# EPICS autosave request: iocBoot/iocLinux/pf4dual.req
$(P)$(H)$(F)bankA
$(P)$(H)$(F)bankB
$(P)$(H)$(F)Z4A
$(P)$(H)$(F)Z3A
$(P)$(H)$(F)Z2A
$(P)$(H)$(F)Z1A
$(P)$(H)$(F)f4A
$(P)$(H)$(F)f3A
$(P)$(H)$(F)f2A
$(P)$(H)$(F)f1A
$(P)$(H)$(F)fPosA
$(P)$(H)$(F)Z4B
$(P)$(H)$(F)Z3B
$(P)$(H)$(F)Z2B
$(P)$(H)$(F)Z1B
$(P)$(H)$(F)f4B
$(P)$(H)$(F)f3B
$(P)$(H)$(F)f2B
$(P)$(H)$(F)f1B
$(P)$(H)$(F)fPosB
$(P)$(H)$(F)useMono
$(P)$(H)$(F)E_using
